// TwinCAT 3 PLC project PLC
// ProgramVersion: 3.1.4026.25
// libraries:
//   Tc2_MC2, * (Beckhoff Automation GmbH)
//   Tc2_Standard, * (Beckhoff Automation GmbH)
//   Tc2_System, * (Beckhoff Automation GmbH)
// project tree:
//   FBs/ DriveBase.TcPOU
//   FBs/Extended/ Drive1.TcPOU, Drive2.TcPOU (not stored)
//   GVLs/ GVL_Eixos.TcGVL
//   ITFs/ I_DriveBase.TcIO
//   / PlcTask.TcTTO
//   POUs/ Habilita_Eixo.TcPOU, MAIN.TcPOU

CONFIGURATION PLC
    RESOURCE PLC ON TwinCAT3
        TASK PlcTask(INTERVAL := T#10ms, PRIORITY := 20);
        PROGRAM MAIN WITH PlcTask : MAIN;
    END_RESOURCE
END_CONFIGURATION

// ---- GVLs/GVL_Eixos.TcGVL
{attribute 'qualified_only'}
VAR_GLOBAL
	Eixo1 : AXIS_REF;
	Eixo2 : AXIS_REF;
END_VAR

// ---- ITFs/I_DriveBase.TcIO
INTERFACE I_DriveBase

METHOD Disable : BOOL
VAR_INPUT
END_VAR
END_METHOD

METHOD Enable : BOOL
VAR_INPUT
END_VAR
END_METHOD

END_INTERFACE

// ---- POUs/MAIN.TcPOU
PROGRAM MAIN
VAR
	
END_VAR

Habilita_Eixo();

END_PROGRAM

// ---- POUs/Habilita_Eixo.TcPOU
PROGRAM Habilita_Eixo
VAR
	DriveMesa: Drive1;
	DriveFuso: Drive2;
	DriveBase: I_DriveBase;
	
	UsarMesa: BOOL;
	UsarFuso: BOOL;
	
END_VAR

IF UsarMesa THEN
	UsarMesa := FALSE;
	DriveBase := DriveMesa;
END_IF

IF DriveFuso THEN
	DriveFuso := FALSE;
	DriveBase := DriveFuso;
END_IF

GVL_Eixos.Eixo1.ReadStatus();
GVL_Eixos.Eixo2.ReadStatus();

DriveBase.Enable();

END_PROGRAM

// ---- FBs/Extended/Drive1.TcPOU
FUNCTION_BLOCK Drive1 EXTENDS DriveBase
VAR_INPUT
END_VAR
VAR_OUTPUT
END_VAR
VAR
END_VAR

{error 'Add method implementation or delete method to use base implementation'}
METHOD Disable : BOOL
END_METHOD

{error 'Add method implementation or delete method to use base implementation'}
METHOD Enable : BOOL
END_METHOD

END_FUNCTION_BLOCK

// ---- FBs/DriveBase.TcPOU
FUNCTION_BLOCK DriveBase IMPLEMENTS I_DriveBase
VAR_INPUT
END_VAR
VAR_OUTPUT
END_VAR
VAR
END_VAR

{warning 'Add method implementation '}
METHOD Disable : BOOL
END_METHOD

METHOD Enable : BOOL

VAR
	MaquinaLigada: BOOL;
	bHabilita: BOOL;
	fb_Habilita1: MC_Power;
END_VAR
IF MaquinaLigada THEN
		bHabilita := 1;
	ELSE
		bHabilita := 0;
	END_IF
	fb_Habilita1(
		Axis:= GVL_Eixos.Eixo1, 
		Enable:= bHabilita, 
		Enable_Positive:= bHabilita, 
		Enable_Negative:= bHabilita, 
		Override:= 100.0);
END_METHOD

END_FUNCTION_BLOCK
